// TIA Portal V16 export
// export: Created 2024-12-03T15:41:41.1081023Z, ExportSetting WithDefaults, DisplayName Totally Integrated Automation Portal, DisplayVersion V16 Update 6, DisplayName TIA Portal Version Control Interface, DisplayVersion V16 Update 2, DisplayName TIA Portal Openness, DisplayVersion V16 Update 6, DisplayName TIA Portal Teamcenter Gateway, DisplayVersion V16, DisplayName SINAMICS Startdrive Advanced, DisplayVersion V16 Update 5, DisplayName SINAMICS Startdrive G130, G150, S120, S150, SINAMICS MV, S210, DisplayVersion V16 Update 5, DisplayName SINAMICS Startdrive G110M, G120, G120C, G120D, G120P, G115D, DisplayVersion V16 Update 5, DisplayName STEP 7 Professional, DisplayVersion V16 Update 6, DisplayName STEP 7 Safety, DisplayVersion V16, DisplayName WinCC Advanced / Unified PC, DisplayVersion V16 Update 6
FUNCTION_BLOCK "AanalogSensor"   // FB44, SCL
{ S7_Optimized_Access := 'FALSE' }
VERSION : 0.1
// stored: AutoNumber true, IsIECCheckEnabled false, SetENOAutomatically false, UDAEnableTagReadback false
   VAR_INPUT
      RawData : Int;
      I_MinRawValue : Int;
      I_MaxRawValue : Int := 1000;
      I_MaxMeasureValue : Real := 100.0;
      I_MinMeasureValue : Real := 0.0;
   END_VAR
   VAR_OUTPUT
      O_ScaledData : Real;
   END_VAR
   VAR_TEMP
      T_NormalizedValue : Real;
   END_VAR
BEGIN
       #T_NormalizedValue := NORM_X_REAL(MIN:=#I_MinRawValue, VALUE:=#RawData, MAX:=#I_MaxRawValue);
       #O_ScaledData := SCALE_X_REAL(MIN:= #I_MinMeasureValue,MAX:= #I_MaxMeasureValue,VALUE := #T_NormalizedValue);
END_FUNCTION_BLOCK
